FUNCTION_BLOCK E_SPLIT_2 (* Split one event into two events *)
  (* Standard: 61499-1 Annex A; Classification: event function block; Function: When EI is Triggered, A Event EO1 followed by a Event EO2 is issued.; Description: Copyright (c) 2017 fortiss GmbH This program and the accompanying materials are made available under the terms of the Eclipse Public License 2.0 which is available at https://www.eclipse.org/legal/epl-2.0/ SPDX-License-Identifier: EPL-2.0 *)
  (* Version 1.0, 2017, Alois Zoitl, fortiss GmbH, initial API and implementation and/or initial documentation *)
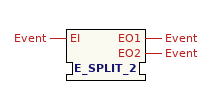
  EVENT_INPUT
    EI; (* Input event *)
  END_EVENT
  EVENT_OUTPUT
    EO1; (* First output event *)
    EO2; (* Second output event *)
  END_EVENT
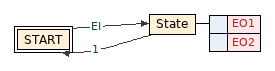
  EC_STATES
    START; (* Initial State *)
    State : -> EO1, -> EO2; (* Output events *)
  END_STATES
  EC_TRANSITIONS
    START TO State := EI;
    State TO START := 1;
  END_TRANSITIONS
END_FUNCTION_BLOCK
